TEXTLIST EL2809_S_1
  1 = 'W circulation pump 1' | chinese: '二级墨盒白循环泵1' | Chinese: '二级墨盒白循环泵1'
  2 = 'W circulation pump 2' | chinese: '二级墨盒白循环泵2' | Chinese: '二级墨盒白循环泵2'
  3 = 'Purge Valve' | chinese: '正压电磁阀' | Chinese: '正压电磁阀'
  4 = 'Vacuum Valve White' | chinese: '负压电磁阀白' | Chinese: '负压电磁阀白'
  5 = 'Vacuum Valve Colcor' | chinese: '负压电磁阀彩' | Chinese: '负压电磁阀彩'
  6 = 'Test piece of power' | chinese: '探块电源' | Chinese: '探块电源'
  7 = ''
  8 = ''
  9 = ''
  10 = ''
  11 = ''
  12 = ''
  13 = ''
  14 = ''
  15 = ''
  16 = ''
   = ''
END_TEXTLIST

(* stored: Version 1.1.0.1, ProductVersion 3.1.4024.11
   TextList EL2809_S_1: Id {97f712fb-ac0e-4076-81c3-8af984bd5c53} *)
